// TIA Portal project "POC_RL_Logic_Controller" (V17)

(* hardware
DEVICE "S7-1500/ET200MP station_1"  S7-1500 station
   slot 0: "Rail_0"  Rack  6ES7 590-1***0-0AA0
   slot 1: "PLC_1"  CPU 1518-4 PN/DP  6ES7 518-4AP00-0AB0  V2.9
      slot 3: "CPU display_1"  6ES7591-1BA00-0AA0
      slot 32768: "PROFINET interface_1"  X1
         slot 32769: "Port_1"  X1 P1
         slot 32770: "Port_2"  X1 P2
      slot 33024: "PROFINET interface_2"  X2
         slot 33025: "Port_1"  X2 P1
      slot 33280: "PROFINET interface GBIT_3"  X3
         slot 33281: "Port_1"  X3 P1
      slot 33536: "DP interface_1"  X4
      slot 34817: "Virtual CP interface port_1"  Virtual CP interface port  Virtual CP interface port
   slot 2: "DI 16x24VDC / DQ 16x24VDC/0.5A BA_1"  DI 16x24VDC/DQ 16x24VDC/0.5A BA  6ES7 523-1BL00-0AA0  V1.1
*)

// ===== PLC "PLC_1"  CPU 1518-4 PN/DP =====

VAR_GLOBAL   // PLC tag table "Default tag table"
   "Grab" AT %Q0.0 : Bool;
   "Conv1" AT %Q0.1 : Bool;
   "Conv2" AT %Q0.2 : Bool;
   "CCW" AT %Q0.3 : Bool;
   "MoveX" AT %Q0.4 : Bool;
   "MoveZ" AT %Q0.5 : Bool;
   "CW" AT %Q0.6 : Bool;
   "Output_Conv" AT %Q0.7 : Bool;
   "Feeding1" AT %Q1.0 : Bool;
   "Feeding2" AT %Q1.1 : Bool;
   "GripperCCW" AT %Q1.2 : Bool;
   "movingX" AT %I0.0 : Bool;
   "movingZ" AT %I0.1 : Bool;
   "wait1" AT %I0.2 : Bool;
   "wait2" AT %I0.3 : Bool;
   "debut_arrivee1" AT %I0.4 : Bool;
   "debut_arrivee2" AT %I0.5 : Bool;
   "rotating" AT %I0.6 : Bool;
   "sortie_piece" AT %I0.7 : Bool;
   "detected" AT %I1.0 : Bool;
   "p_exit" AT %I1.1 : Bool;
   "init" AT %I1.2 : Bool;
END_VAR

DATA_BLOCK "Control Table"   // DB1
{ S7_Optimized_Access := 'TRUE' }
VERSION : 0.1
   VAR
      State : Array[0..235] of DInt;
      Action : Array[0..235] of Int;
   END_VAR
BEGIN
   State[1] := 3528021;
   State[2] := 5592151;
   State[3] := 5592407;
   State[4] := 5594613;
   State[5] := 5594869;
   State[6] := 5723477;
   State[7] := 6116693;
   State[8] := 7705941;
   State[9] := 7722325;
   State[10] := 9789141;
   State[11] := 9789397;
   State[12] := 9794901;
   State[13] := 9917781;
   State[14] := 10310997;
   State[15] := 11883605;
   State[16] := 11883861;
   State[17] := 13976661;
   State[18] := 13988949;
   State[19] := 13989205;
   State[20] := 14112085;
   State[21] := 16078165;
   State[22] := 18174805;
   State[23] := 18175069;
   State[24] := 18175325;
   State[25] := 18177525;
   State[26] := 18183509;
   State[27] := 18306389;
   State[28] := 19256661;
   State[29] := 20305237;
   State[30] := 20305493;
   State[31] := 21321045;
   State[32] := 22304085;
   State[33] := 22304597;
   State[34] := 22306805;
   State[35] := 22353237;
   State[36] := 22368341;
   State[37] := 22368343;
   State[38] := 22369109;
   State[39] := 22369111;
   State[40] := 22369301;
   State[41] := 22369349;
   State[42] := 22369361;
   State[43] := 22369364;
   State[44] := 22369367;
   State[45] := 22369373;
   State[46] := 22369617;
   State[47] := 22369620;
   State[48] := 22369623;
   State[49] := 22369629;
   State[50] := 22369813;
   State[51] := 22369879;
   State[52] := 22369885;
   State[53] := 22370069;
   State[54] := 22370117;
   State[55] := 22370129;
   State[56] := 22370135;
   State[57] := 22370141;
   State[58] := 22370805;
   State[59] := 22371317;
   State[60] := 22371573;
   State[61] := 22371813;
   State[62] := 22371829;
   State[63] := 22372085;
   State[64] := 22372277;
   State[65] := 22372325;
   State[66] := 22372341;
   State[67] := 22373717;
   State[68] := 22377813;
   State[69] := 22500693;
   State[70] := 22631765;
   State[71] := 23450965;
   State[72] := 23451221;
   State[73] := 24483157;
   State[74] := 24499285;
   State[75] := 24499541;
   State[76] := 25515349;
   State[77] := 25515861;
   State[78] := 26498389;
   State[79] := 26498901;
   State[80] := 26501077;
   State[81] := 26559829;
   State[82] := 26562645;
   State[83] := 26563413;
   State[84] := 26563677;
   State[85] := 26563921;
   State[86] := 26563933;
   State[87] := 26564189;
   State[88] := 26564373;
   State[89] := 26564433;
   State[90] := 26564445;
   State[91] := 26565333;
   State[92] := 26565589;
   State[93] := 26565845;
   State[94] := 26566101;
   State[95] := 26566357;
   State[96] := 26566549;
   State[97] := 26566613;
   State[98] := 26568021;
   State[99] := 26571861;
   State[100] := 26572117;
   State[101] := 26694741;
   State[102] := 26694997;
   State[103] := 26826069;
   State[104] := 27612245;
   State[105] := 27612501;
   State[106] := 27613013;
   State[107] := 28660821;
   State[108] := 28661077;
   State[109] := 28661333;
   State[110] := 28661589;
   State[111] := 29709653;
   State[112] := 30692693;
   State[113] := 30693205;
   State[114] := 30695381;
   State[115] := 30753877;
   State[116] := 30754133;
   State[117] := 30756949;
   State[118] := 30757461;
   State[119] := 30758225;
   State[120] := 30758228;
   State[121] := 30758237;
   State[122] := 30759637;
   State[123] := 30760661;
   State[124] := 30760917;
   State[125] := 30762069;
   State[126] := 30762325;
   State[127] := 30766165;
   State[128] := 30766421;
   State[129] := 30889045;
   State[130] := 30889301;
   State[131] := 31806805;
   State[132] := 32855125;
   State[133] := 32855381;
   State[134] := 34954869;
   State[135] := 34955125;
   State[136] := 34985045;
   State[137] := 34985301;
   State[138] := 35083605;
   State[139] := 35476821;
   State[140] := 38884693;
   State[141] := 39081301;
   State[142] := 39081813;
   State[143] := 39083893;
   State[144] := 39145557;
   State[145] := 39145559;
   State[146] := 39146325;
   State[147] := 39146327;
   State[148] := 39146583;
   State[149] := 39146836;
   State[150] := 39146839;
   State[151] := 39148405;
   State[152] := 39148661;
   State[153] := 39148917;
   State[154] := 39149157;
   State[155] := 39149173;
   State[156] := 39149413;
   State[157] := 39149429;
   State[158] := 39163221;
   State[159] := 39179349;
   State[160] := 39179605;
   State[161] := 39179861;
   State[162] := 39277653;
   State[163] := 39277909;
   State[164] := 39408981;
   State[165] := 39670869;
   State[166] := 39671125;
   State[167] := 43078997;
   State[168] := 43337045;
   State[169] := 43340629;
   State[170] := 43340885;
   State[171] := 43341141;
   State[172] := 43341653;
   State[173] := 43342677;
   State[174] := 43342933;
   State[175] := 43343189;
   State[176] := 43343445;
   State[177] := 43343701;
   State[178] := 43349077;
   State[179] := 43349333;
   State[180] := 43471957;
   State[181] := 43472213;
   State[182] := 43865173;
   State[183] := 43865429;
   State[184] := 47469909;
   State[185] := 47470421;
   State[186] := 47472469;
   State[187] := 47531093;
   State[188] := 47531349;
   State[189] := 47535444;
   State[190] := 47535445;
   State[191] := 47537749;
   State[192] := 47538005;
   State[193] := 47539285;
   State[194] := 47539541;
   State[195] := 47543381;
   State[196] := 47543637;
   State[197] := 47666517;
   State[198] := 51762517;
   State[199] := 51860821;
   State[200] := 51991893;
   State[201] := 52253781;
   State[202] := 52254037;
   State[203] := 55661653;
   State[204] := 55661909;
   State[205] := 55858517;
   State[206] := 55907669;
   State[207] := 55923793;
   State[208] := 55924049;
   State[209] := 55924055;
   State[210] := 55940437;
   State[211] := 55956821;
   State[212] := 56055125;
   State[213] := 56185941;
   State[214] := 56186197;
   State[215] := 56448085;
   State[216] := 56448341;
   State[217] := 59855957;
   State[218] := 59856213;
   State[219] := 60052821;
   State[220] := 60053333;
   State[221] := 60055381;
   State[222] := 60118353;
   State[223] := 60118357;
   State[224] := 60118865;
   State[225] := 60120917;
   State[226] := 60249173;
   State[227] := 60249429;
   State[228] := 60380245;
   State[229] := 60380501;
   State[230] := 60642389;
   State[231] := 60642645;
   State[232] := 60642901;
   State[233] := 60643153;
   State[234] := 64312661;
   State[235] := 67108865;
   Action[0] := 2;
   Action[2] := 13;
   Action[3] := 13;
   Action[4] := 11;
   Action[6] := 5;
   Action[7] := 4;
   Action[9] := 3;
   Action[10] := 8;
   Action[11] := 10;
   Action[12] := 7;
   Action[13] := 5;
   Action[14] := 4;
   Action[15] := 3;
   Action[16] := 3;
   Action[18] := 2;
   Action[19] := 7;
   Action[20] := 5;
   Action[21] := 3;
   Action[23] := 12;
   Action[24] := 12;
   Action[25] := 8;
   Action[26] := 7;
   Action[27] := 5;
   Action[29] := 6;
   Action[30] := 3;
   Action[38] := 9;
   Action[39] := 9;
   Action[44] := 13;
   Action[45] := 12;
   Action[48] := 13;
   Action[49] := 12;
   Action[53] := 9;
   Action[54] := 9;
   Action[55] := 9;
   Action[56] := 9;
   Action[57] := 12;
   Action[59] := 9;
   Action[60] := 11;
   Action[62] := 8;
   Action[63] := 11;
   Action[64] := 9;
   Action[65] := 9;
   Action[66] := 9;
   Action[68] := 7;
   Action[69] := 5;
   Action[74] := 6;
   Action[75] := 3;
   Action[77] := 9;
   Action[84] := 12;
   Action[86] := 12;
   Action[87] := 12;
   Action[88] := 9;
   Action[90] := 9;
   Action[92] := 9;
   Action[93] := 10;
   Action[94] := 8;
   Action[95] := 10;
   Action[96] := 9;
   Action[97] := 9;
   Action[99] := 7;
   Action[100] := 7;
   Action[102] := 5;
   Action[107] := 3;
   Action[108] := 3;
   Action[109] := 3;
   Action[110] := 9;
   Action[111] := 2;
   Action[112] := 2;
   Action[113] := 2;
   Action[114] := 2;
   Action[115] := 2;
   Action[119] := 2;
   Action[121] := 12;
   Action[123] := 8;
   Action[124] := 9;
   Action[125] := 2;
   Action[126] := 2;
   Action[127] := 7;
   Action[128] := 7;
   Action[129] := 2;
   Action[130] := 5;
   Action[133] := 2;
   Action[134] := 11;
   Action[135] := 11;
   Action[137] := 6;
   Action[139] := 4;
   Action[146] := 9;
   Action[147] := 9;
   Action[148] := 13;
   Action[150] := 13;
   Action[151] := 9;
   Action[152] := 11;
   Action[155] := 11;
   Action[156] := 9;
   Action[157] := 9;
   Action[159] := 6;
   Action[160] := 6;
   Action[163] := 5;
   Action[165] := 4;
   Action[166] := 4;
   Action[169] := 9;
   Action[172] := 9;
   Action[173] := 9;
   Action[175] := 8;
   Action[176] := 8;
   Action[177] := 9;
   Action[178] := 7;
   Action[179] := 7;
   Action[181] := 5;
   Action[183] := 4;
   Action[185] := 2;
   Action[187] := 2;
   Action[188] := 2;
   Action[190] := 2;
   Action[191] := 2;
   Action[192] := 9;
   Action[193] := 2;
   Action[194] := 2;
   Action[195] := 7;
   Action[196] := 7;
   Action[197] := 5;
   Action[198] := 1;
   Action[199] := 1;
   Action[201] := 4;
   Action[202] := 1;
   Action[203] := 1;
   Action[204] := 1;
   Action[205] := 1;
   Action[209] := 1;
   Action[210] := 1;
   Action[211] := 1;
   Action[212] := 5;
   Action[213] := 1;
   Action[214] := 1;
   Action[215] := 1;
   Action[216] := 4;
   Action[217] := 1;
   Action[218] := 1;
   Action[219] := 1;
   Action[220] := 1;
   Action[223] := 1;
   Action[225] := 1;
   Action[227] := 5;
   Action[228] := 1;
   Action[229] := 1;
   Action[230] := 4;
   Action[231] := 4;
   Action[233] := 9;
   Action[234] := 2;
END_DATA_BLOCK

DATA_BLOCK "State_Action_DB"   // DB2
{ S7_Optimized_Access := 'TRUE' }
VERSION : 0.1
// stored: InstanceOfName BinarySearch
"BinarySearch"
BEGIN
END_DATA_BLOCK

DATA_BLOCK "Program_DB"   // DB10
{ S7_Optimized_Access := 'TRUE' }
VERSION : 0.1
// stored: InstanceOfName Program
"Program"
BEGIN
END_DATA_BLOCK

FUNCTION_BLOCK "BinarySearch"   // FB1, SCL
{ S7_Optimized_Access := 'TRUE' }
VERSION : 0.1
   VAR_INPUT
      S_State : DInt;
   END_VAR
   VAR_OUTPUT
      Action : Int;
   END_VAR
   VAR_IN_OUT
      ArEtat : Array[*] of DInt;
      ArAction : Array[*] of Int;
   END_VAR
   VAR_TEMP
      max : DInt;
      min : DInt;
      mid : DInt;
   END_VAR
BEGIN
   #min := 0;
   #max:=UPPER_BOUND(ARR := #ArEtat, DIM := 1);

   WHILE #min < #max DO
       #mid := (#min + #max) / 2;
       IF  #ArEtat[#mid] = #S_State THEN
           #Action := #ArAction[#mid];
           RETURN
           ;
       ELSIF  #ArEtat[#mid] < #S_State THEN
           #min := #mid + 1;
       ELSE
           #max := #mid - 1;
       END_IF;

   END_WHILE;

   IF #ArEtat[#min] = #S_State THEN
       #Action := #ArAction[#min];
       RETURN;
   ELSE
       #Action := 0;
       RETURN;
   END_IF;
END_FUNCTION_BLOCK

FUNCTION_BLOCK "Program"   // FB2, SCL
{ S7_Optimized_Access := 'TRUE' }
VERSION : 0.1
   VAR
      task : Array[0..13] of Struct
         AUT : Bool;
         AUTf : Bool;
         IC : Bool;
         IS : Bool;
      END_STRUCT;
      FTX10 : Bool;
      FTX11 : Bool;
      FTX20 : Bool;
      FTX21 : Bool;
      FTX30 : Bool;
      FTX31 : Bool;
      FTX40 : Bool;
      FTX41 : Bool;
      FTX50 : Bool;
      FTX51 : Bool;
      FTX52 : Bool;
      FTX53 : Bool;
      FTX54 : Bool;
      FTX55 : Bool;
      FTX60 : Bool;
      FTX61 : Bool;
      FTX70 : Bool;
      FTX71 : Bool;
      FTX80 : Bool;
      FTX81 : Bool;
      FTX82 : Bool;
      FTX83 : Bool;
      FTX90 : Bool;
      FTX91 : Bool;
      FTX100 : Bool;
      FTX101 : Bool;
      FTX110 : Bool;
      FTX111 : Bool;
      FTX120 : Bool;
      FTX121 : Bool;
      FTX122 : Bool;
      FTX123 : Bool;
      FTX130 : Bool;
      FTX131 : Bool;
      FTX132 : Bool;
      FTX133 : Bool;
      position : Real;
      X10 : Bool;
      X11 : Bool;
      X20 : Bool;
      X21 : Bool;
      X30 : Bool;
      X31 : Bool;
      X40 : Bool;
      X41 : Bool;
      X50 : Bool;
      X51 : Bool;
      X52 : Bool;
      X53 : Bool;
      X54 : Bool;
      X55 : Bool;
      X60 : Bool;
      X61 : Bool;
      X70 : Bool;
      X71 : Bool;
      X80 : Bool;
      X81 : Bool;
      X82 : Bool;
      X83 : Bool;
      X90 : Bool;
      X91 : Bool;
      X100 : Bool;
      X101 : Bool;
      X110 : Bool;
      X111 : Bool;
      X120 : Bool;
      X121 : Bool;
      X122 : Bool;
      X123 : Bool;
      X130 : Bool;
      X131 : Bool;
      X132 : Bool;
      X133 : Bool;
      retracted : Bool;
      sorti : Bool;
      up : Bool;
      bas : Bool;
      i : Int;
      State : DInt;
      ActionFound : Int;
   END_VAR
BEGIN
   "R_TRIG_movingX"(CLK := "movingX");
   "R_TRIG_movingZ"(CLK := "movingZ");
   "R_TRIG_rotating"(CLK := "rotating");

   "F_TRIG_movingX"(CLK := "movingX");
   "F_TRIG_movingZ"(CLK := "movingZ");
   "F_TRIG_rotating"(CLK := "rotating");
   "F_TRIG_sortie_piece"(CLK := "sortie_piece");

   IF "init" THEN
       #up := True;
       #bas := False;
       #retracted := True;
       #sorti := False;
       "MoveX" := False;
       "MoveZ" := False;
       "CCW" := False;
       "CW" := False;
       "Grab" := False;
       "Conv1" := False;
       "Conv2" := False;
       "Output_Conv" := False;
       "GripperCCW" := False;
       #position := 0;
   END_IF;


   IF "MoveX" AND "R_TRIG_movingX".Q THEN
       #retracted := False;
       #sorti := False;
   END_IF;
   IF "MoveX" AND "F_TRIG_movingX".Q THEN
       #retracted := False;
       #sorti := True;
   END_IF;
   IF NOT "MoveX" AND "R_TRIG_movingX".Q THEN
       #retracted := False;
       #sorti := False;
   END_IF;
   IF NOT "MoveX" AND "F_TRIG_movingX".Q THEN
       #retracted := True;
       #sorti := False;
   END_IF;
   IF "MoveZ" AND "R_TRIG_movingZ".Q THEN
       #up := False;
       #bas := False;
   END_IF;
   IF "MoveZ" AND "F_TRIG_movingZ".Q THEN
       #up := False;
       #bas := True;
   END_IF;
   IF NOT "MoveZ" AND "R_TRIG_movingZ".Q THEN
       #up := False;
       #bas := False;
   END_IF;
   IF NOT "MoveZ" AND "F_TRIG_movingZ".Q THEN
       #up := True;
       #bas := False;
   END_IF;

   #task[1].IS := #X10;
   #task[2].IS := #X20;
   #task[3].IS := #X30;
   #task[4].IS := #X40;
   #task[5].IS := #X50;
   #task[6].IS := #X60;
   #task[7].IS := #X70;
   #task[8].IS := #X80;
   #task[9].IS := #X90;
   #task[10].IS := #X100;
   #task[11].IS := #X110;
   #task[12].IS := #X120;
   #task[13].IS := #X130;

   #task[1].IC := NOT "wait1";
   #task[2].IC := NOT "wait2";
   #task[3].IC := (#position = 0) AND #retracted AND "wait1" AND #up AND NOT "detected";
   #task[4].IC := #up AND #retracted AND "detected" AND (#position = 1);
   #task[5].IC := #up AND #retracted AND "detected" AND (#position = 2);
   #task[6].IC := (#position = 0) AND #retracted AND "wait2" AND #up AND NOT "detected";
   #task[7].IC := #up AND #retracted AND "detected" AND (#position = 3);
   #task[8].IC := #up AND #retracted AND NOT "detected" AND (#position = 2);
   #task[9].IC := "p_exit";
   #task[10].IC := (#position = 2) AND #retracted AND #up AND NOT "detected" AND "wait1";
   #task[11].IC := (#position = 2) AND #retracted AND #up AND NOT "detected" AND "wait2";
   #task[12].IC := #retracted AND "wait1" AND #up AND NOT "detected" AND (#position = 1);
   #task[13].IC := #retracted AND "wait2" AND #up AND NOT "detected" AND (#position = 3);

   #State := 0;
   FOR #i := 0 TO 13 DO
       #State := #State + BOOL_TO_INT(#task[13-#i].IS) * 2 ** (#i * 2);
       #State := #State + BOOL_TO_INT(#task[13-#i].IC) * 2 ** ((#i * 2) + 1);
   END_FOR;

   "State_Action_DB"(S_State:=#State,
                     Action=>#ActionFound,
                     ArEtat:="Control Table".State,
                     ArAction:="Control Table".Action);


   FOR #i := 0 TO 13 DO
       #task[#i].AUTf := 0;
   END_FOR;
   #task[#ActionFound].AUTf := 1;

   #task[1].AUT := #task[12].IS AND #task[1].AUTf;
   #task[2].AUT := #task[13].IS AND #task[2].AUTf;
   #task[3].AUT := #task[6].IS AND #task[3].AUTf;
   #task[4].AUT := #task[12].IS AND #task[4].AUTf;
   #task[5].AUT := #task[8].IS AND #task[9].IS AND #task[10].IS AND #task[11].IS AND #task[5].AUTf;
   #task[6].AUT := #task[3].IS AND #task[6].AUTf;
   #task[7].AUT := #task[8].IS AND #task[13].IS AND #task[7].AUTf;
   #task[8].AUT := #task[5].IS AND #task[7].IS AND #task[10].IS AND #task[11].IS AND #task[8].AUTf;
   #task[9].AUT := #task[5].IS AND #task[9].AUTf;
   #task[10].AUT := #task[5].IS AND #task[8].IS AND #task[11].IS AND #task[10].AUTf;
   #task[11].AUT := #task[5].IS AND #task[8].IS AND #task[10].IS AND #task[11].AUTf;
   #task[12].AUT := #task[1].IS AND #task[4].IS AND #task[8].IS AND #task[12].AUTf;
   #task[13].AUT := #task[2].IS AND #task[7].IS AND #task[8].IS AND #task[13].AUTf;

   (*Transition : GConv1_T1*)
   #FTX10 := #task[1].IS AND #task[1].AUT AND #task[1].IC;
   #FTX11 := #X11 AND "wait1";

   (*Transition : GConv2_T2*)
   #FTX20 := #X20 AND #task[2].AUT AND #task[2].IC;
   #FTX21 := #X21 AND "wait2";

   (* Transition : GCCW0_1_T3*)
   #FTX30 := #X30 AND #task[3].AUT AND #task[3].IC;
   #FTX31 := #X31 AND "F_TRIG_rotating".Q;

   (* Transition : GCCW1_2_T4*)
   #FTX40 := #X40 AND #task[4].AUT AND #task[4].IC;
   #FTX41 := #X41 AND "F_TRIG_rotating".Q;

   (* Transition : GDEPOSER_T5*)
   #FTX50 := #X50 AND #task[5].AUT AND #task[5].IC;
   #FTX51 := #X51 AND "F_TRIG_movingX".Q;
   #FTX52 := #X52 AND "F_TRIG_movingZ".Q;
   #FTX53 := #X53;
   #FTX54 := #X54 AND "F_TRIG_movingZ".Q;
   #FTX55 := #X55 AND "F_TRIG_movingX".Q;

   (* Transition : GCW0_3_T6*)
   #FTX60 := #X60 AND #task[6].AUT AND #task[6].IC;
   #FTX61 := #X61 AND "F_TRIG_rotating".Q;

   (* Transition : GCW3_2_T7*)
   #FTX70 := #X70 AND #task[7].AUT AND #task[7].IC;
   #FTX71 := #X71 AND "F_TRIG_rotating".Q;

   (* Transition : GCCW2_0_T8*)
   #FTX80 := #X80 AND #task[8].AUT AND #task[8].IC;
   #FTX81 := #X81 AND "F_TRIG_rotating".Q;
   #FTX82 := #X82;
   #FTX83 := #X83 AND "F_TRIG_rotating".Q;

   (* Transition : GConv_Sortie_T9*)
   #FTX90 := #X90 AND #task[9].AUT AND #task[9].IC;
   #FTX91 := #X91 AND "F_TRIG_sortie_piece".Q;

   (* Transition : GCW3_2_T10*)
   #FTX100 := #X100 AND #task[10].AUT AND #task[10].IC;
   #FTX101 := #X101 AND "F_TRIG_rotating".Q;

   (* Transition : GCCW2_3_T11*)
   #FTX110 := #X110 AND #task[11].AUT AND #task[11].IC;
   #FTX111 := #X111 AND "F_TRIG_rotating".Q;

   (* Transition : GPRENDRE_1_T12*)
   #FTX120 := #X120 AND #task[12].AUT AND #task[12].IC;
   #FTX121 := #X121 AND "F_TRIG_movingZ".Q;
   #FTX122 := #X122;
   #FTX123 := #X123 AND "F_TRIG_movingZ".Q;

   (* Transition : GPRENDRE_2_T13*)
   #FTX130 := #X130 AND #task[13].AUT AND #task[13].IC;
   #FTX131 := #X131 AND "F_TRIG_movingZ".Q;
   #FTX132 := #X132;
   #FTX133 := #X133 AND "F_TRIG_movingZ".Q;

   IF "CCW" AND "R_TRIG_rotating".Q THEN
       #position := #position + 0.5;
   END_IF;
   IF (#X31 OR #X41 OR #X81 OR #X83 OR #X111) AND "F_TRIG_rotating".Q THEN
       #position := #position + 0.5;
   END_IF;

   IF "CW" AND "R_TRIG_rotating".Q THEN
       #position := #position - 0.5;
   END_IF;
   IF (#X61 OR #X71 OR #X101) AND "F_TRIG_rotating".Q THEN
       #position := #position - 0.5;
   END_IF;

   IF #position = 4 THEN
       #position := 0;
   END_IF;
   IF #position < 0 THEN
       #position := 3.5;
   END_IF;

   (*# Task 1 : GConv1_T1*)
   #X10 := #FTX11 OR #X10 AND NOT #FTX10 OR "init";
   #X11 := (#FTX10 OR #X11 AND NOT #FTX11) AND NOT "init";

   (*# Etape : GConv2_T2*)
   #X20 := #FTX21 OR #X20 AND NOT #FTX20 OR "init";
   #X21 := (#FTX20 OR #X21 AND NOT #FTX21) AND NOT "init";

   (*# Etape : GCCW0_1_T3*)
   #X30 := #FTX31 OR #X30 AND NOT #FTX30 OR "init";
   #X31 := (#FTX30 OR #X31 AND NOT #FTX31) AND NOT "init";

   (*# Etape : GCCW1_2_T4*)
   #X40 := #FTX41 OR #X40 AND NOT #FTX40 OR "init";
   #X41 := (#FTX40 OR #X41 AND NOT #FTX41) AND NOT "init";

   (*# Etape : GDEPOSER_T5*)
   #X50 := #FTX55 OR #X50 AND NOT #FTX50 OR "init";
   #X51 := (#FTX50 OR #X51 AND NOT #FTX51) AND NOT "init";
   #X52 := (#FTX51 OR #X52 AND NOT #FTX52) AND NOT "init";
   #X53 := (#FTX52 OR #X53 AND NOT #FTX53) AND NOT "init";
   #X54 := (#FTX53 OR #X54 AND NOT #FTX54) AND NOT "init";
   #X55 := (#FTX54 OR #X55 AND NOT #FTX55) AND NOT "init";

   (*# Etape : GCW0_3_T6*)
   #X60 := #FTX61 OR #X60 AND NOT #FTX60 OR "init";
   #X61 := (#FTX60 OR #X61 AND NOT #FTX61) AND NOT "init";

   (*# Etape : GCW3_2_T7*)
   #X70 := #FTX71 OR #X70 AND NOT #FTX70 OR "init";
   #X71 := (#FTX70 OR #X71 AND NOT #FTX71) AND NOT "init";

   (*# Etape : GCCW2_0_T8*)
   #X80 := #FTX83 OR #X80 AND NOT #FTX80 OR "init";
   #X81 := (#FTX80 OR #X81 AND NOT #FTX81) AND NOT "init";
   #X82 := (#FTX81 OR #X82 AND NOT #FTX82) AND NOT "init";
   #X83 := (#FTX82 OR #X83 AND NOT #FTX83) AND NOT "init";

   (*# Etape : GConv_Sortie_T9*)
   #X90 := #FTX91 OR #X90 AND NOT #FTX90 OR "init";
   #X91 := (#FTX90 OR #X91 AND NOT #FTX91) AND NOT "init";

   (*# Etape : GCW3_2_T10*)
   #X100 := #FTX101 OR #X100 AND NOT #FTX100 OR "init";
   #X101 := (#FTX100 OR #X101 AND NOT #FTX101) AND NOT "init";

   (*# Etape : GCCW2_3_T11*)
   #X110 := #FTX111 OR #X110 AND NOT #FTX110 OR "init";
   #X111 := (#FTX110 OR #X111 AND NOT #FTX111) AND NOT "init";

   (*# Etape : GPRENDRE_1_T12*)
   #X120 := #FTX123 OR #X120 AND NOT #FTX120 OR "init";
   #X121 := (#FTX120 OR #X121 AND NOT #FTX121) AND NOT "init";
   #X122 := (#FTX121 OR #X122 AND NOT #FTX122) AND NOT "init";
   #X123 := (#FTX122 OR #X123 AND NOT #FTX123) AND NOT "init";

   (*# Etape : GPRENDRE_2_T13*)
   #X130 := #FTX133 OR #X130 AND NOT #FTX130 OR "init";
   #X131 := (#FTX130 OR #X131 AND NOT #FTX131) AND NOT "init";
   #X132 := (#FTX131 OR #X132 AND NOT #FTX132) AND NOT "init";
   #X133 := (#FTX132 OR #X133 AND NOT #FTX133) AND NOT "init";

   (*# Action*)
   IF #FTX52 THEN
       "Grab" := False;
   END_IF;
   IF #FTX121 THEN
       "Grab" := True;
   END_IF;
   IF #FTX131 THEN
       "Grab" := True;
   END_IF;
   "Conv1" := #X11;
   "Conv2" := #X21;
   IF #FTX30 OR #FTX40 OR #FTX80 OR #FTX82 OR #FTX110 THEN
       "CCW" := True;
   END_IF;
   IF (#X31 OR #X41 OR #X81 OR #X83 OR #X111) AND "R_TRIG_rotating".Q THEN
       "CCW" := False;
   END_IF;
   "MoveX" := #X51 OR #X52 OR #X53 OR #X54;
   "MoveZ" := #X52 OR #X53 OR #X121 OR #X122 OR #X131 OR #X132;
   IF #FTX60 OR #FTX70 OR #FTX100 THEN
       "CW" := True;
   END_IF;
   IF (#X61 OR #X71 OR #X101) AND "R_TRIG_rotating".Q THEN
       "CW" := False;
   END_IF;
   "Output_Conv" := #X91;
   "Feeding1" := #X11 OR NOT "debut_arrivee1";
   "Feeding2" := #X21 OR NOT "debut_arrivee2";
   "GripperCCW" := #X51;
END_FUNCTION_BLOCK

ORGANIZATION_BLOCK "Main"   // OB1, LAD, ProgramCycle
TITLE = "Main Program Sweep (Cycle)"
{ S7_Optimized_Access := 'TRUE' }
VERSION : 0.1
   VAR_INPUT
      Initial_Call : Bool;   // Initial call of this OB
      Remanence : Bool;   // =True, if remanent data are available
   END_VAR
BEGIN

REGION Network 1
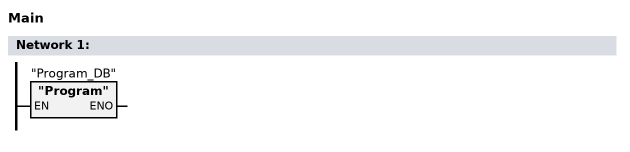
   RUNG wire#powerrail
      "Program_DB"()
   END_RUNG
   // the same network as SCL:
   "Program_DB"();   // "Program"
END_REGION
END_ORGANIZATION_BLOCK